FUNCTION_BLOCK FB_dither
VAR_INPUT
END_VAR
VAR_OUTPUT
END_VAR
VAR
	// dithering signal type
	// 1: square
	m_type:INT := 1;
	
	// dithering amplitude
	m_amplitude:LREAL;
	
	// dithering frequency
	m_frequency :LREAL;
	
	// time step
	m_timeStep :LREAL;
	
	// time period
	m_timePeriod:LREAL:=0.0;
END_VAR

METHOD init : BOOL
VAR_INPUT
	i_type:INT;
	i_timeStep:LREAL;
	i_amp:LREAL;
	i_freq:LREAL;
END_VAR
m_type:=i_type;
m_timeStep:=i_timeStep;
m_amplitude:=i_amp;
m_frequency:= i_freq;
m_timePeriod:=0;
END_METHOD

METHOD run : LREAL
VAR_INPUT
END_VAR
VAR
	tmpVar :LREAL;
END_VAR
m_timePeriod := m_timePeriod+ m_timeStep;
run:=0;

CASE m_type OF
	// sin
	1:
		run := m_amplitude*SIN(2*pi*m_frequency * m_timePeriod);
	// square
	2:
		tmpVar := SIN(2*pi*m_frequency * m_timePeriod);
		run:= sign(tmpVar) * m_amplitude;
	
END_CASE
END_METHOD

END_FUNCTION_BLOCK

(* stored: Version 1.1.0.1, ProductVersion 3.1.4024.11
   POU FB_dither: Id {6027c9a2-000c-4507-99b9-8b28cc54778d}, SpecialFunc None
   Method init: Id {92c8e503-440f-47d0-8384-9bcdedaa4795}
   Method run: Id {99dad32a-86c0-4782-9867-6705f013c06b} *)
